// TIA Portal V17 export
// export: Created 2024-08-07T21:44:00.2293512Z, ExportSetting WithDefaults, DisplayName Totally Integrated Automation Portal, DisplayVersion V17 Update 7, DisplayName TIA Portal Openness, DisplayVersion V17 Update 7, DisplayName TIA Portal Version Control Interface, DisplayVersion V17, DisplayName SINAMICS Startdrive Advanced, DisplayVersion V17 SP2, DisplayName SINAMICS Startdrive G110M, G120, G120C, G120D, G120P, G115D, DisplayVersion V17 SP2, DisplayName SINAMICS Startdrive G130, G150, S120, S150, SINAMICS MV, S210, DisplayVersion V17 SP2, DisplayName STEP 7 Professional, DisplayVersion V17 Update 7, DisplayName STEP 7 Safety, DisplayVersion V17 Update 6, DisplayName WinCC Advanced / Unified PC, DisplayVersion V17 Update 7
DATA_BLOCK "DB_Eks_Instance"   // DB5050
VERSION : 0.1
// stored: AutoNumber false, DBAccessibleFromOPCUA true, DBAccessibleFromWebserver true, InstanceOfName FB_Eks, InstanceOfType FB
"FB_Eks"
   // VAR_INPUT
   //    iScreenNumberEqual : Bool := FALSE;
   //    iOpSwitchManualMode : Bool := TRUE;
   //    iGenerateTimeoutError : Bool := FALSE;
   //    iPermanentAccess : Bool := FALSE;
   //    iBlinker : Bool := TRUE;
   // END_VAR
   // VAR_OUTPUT
   //    qManualModeActive : Bool := TRUE;
   //    qOpManualModeLamp : Bool := TRUE;
   //    qeKeyTimeout : Bool := FALSE;
   // END_VAR
   // VAR
   //    Status : Struct
   //       Key : Struct
   //          Inserted : Bool := TRUE;
   //          Found : Bool := TRUE;
   //          Valid : Bool := TRUE;
   //          ActualKeyStatus : Int := 5;
   //          LastKeyStatus : Int := 0;
   //       END_STRUCT;
   //       Global : Struct
   //          GapLeader : Bool := FALSE;
   //          Maintenance : Bool := FALSE;
   //          Engineer : Bool := TRUE;
   //          MaintenanceOrEngineer : Bool := TRUE;
   //          AnyValidKey : Bool := TRUE;
   //       END_STRUCT;
   //       ManualMode : Struct
   //          GapLeader : Bool := FALSE;
   //          Maintenance : Bool := FALSE;
   //          Engineer : Bool := TRUE;
   //          MaintenanceOrEngineer : Bool := TRUE;
   //          AnyValidKey : Bool := TRUE;
   //       END_STRUCT;
   //    END_STRUCT;
   //    Database : Struct
   //       Status : Struct
   //          ActualAndLastKeyEqual { ExternalAccessible := 'False'; ExternalVisible := 'False'; ExternalWritable := 'False'} : Bool := FALSE;
   //          LastKeyIsEmpty : Bool := FALSE;
   //          LastKeyEmployeeIDIsEmpty : Bool := FALSE;
   //          LastKeyFound { ExternalAccessible := 'False'; ExternalVisible := 'False'; ExternalWritable := 'False'} : Bool := FALSE;
   //          LastKeyIndex { ExternalAccessible := 'False'; ExternalVisible := 'False'; ExternalWritable := 'False'} : Int := 0;
   //          FreePlaceFound { ExternalAccessible := 'False'; ExternalVisible := 'False'; ExternalWritable := 'False'} : Bool := FALSE;
   //          FreePlaceIndex { ExternalAccessible := 'False'; ExternalVisible := 'False'; ExternalWritable := 'False'} : Int := 0;
   //          NumberOfKeys : Int := 100;
   //          NumberOfStoredKeys : Int := 0;
   //          StoredKeysReachedMaximum : Bool := FALSE;
   //          NumberOfEngineerKeys : Int := 50;
   //          NumberOfStoredEngineerKeys : Int := 0;
   //          StoredEngineerKeysReachedMaximum : Bool := FALSE;
   //       END_STRUCT;
   //       ListNumber : Int := 1;
   //       ListNumberLast : Int := 1;
   //    END_STRUCT;
   //    KeyManage : Struct
   //       CanBeAdd : Bool := FALSE;
   //       Add : Bool := FALSE;
   //       CanBeRemoved : Bool := FALSE;
   //       Remove : Bool := FALSE;
   //       CanBeUsed : Bool := FALSE;
   //       Use : Int := 0;
   //       CanBeSearched : Bool := FALSE;
   //       Search : Bool := FALSE;
   //       Searching : Bool := FALSE;
   //       SearchedRow : Int := 0;
   //       SearchedRowHMI : Int := 0;
   //    END_STRUCT;
   // END_VAR
   // VAR RETAIN
   //    KeyTimeout : Time := T#2H_46M_39S;
   // END_VAR
   // VAR
   //    KeyInsertedInReader { S7_SetPoint := 'True'} : R_TRIG;
   //    KeyRemovedFromReader { S7_SetPoint := 'True'} : F_TRIG;
   //    TONs : Struct
   //       tDelayTimeoutError { S7_SetPoint := 'True'} : TON_TIME;
   //    END_STRUCT;
   // END_VAR
BEGIN
   KeyInsertedInReader.CLK := TRUE;
   KeyInsertedInReader.Q := FALSE;
   KeyInsertedInReader.Stat_Bit := TRUE;
   KeyRemovedFromReader.CLK := TRUE;
   KeyRemovedFromReader.Q := FALSE;
   KeyRemovedFromReader.Stat_Bit := TRUE;
   TONs.tDelayTimeoutError.PT := T#0MS;
   TONs.tDelayTimeoutError.IN := FALSE;
END_DATA_BLOCK
